FUNCTION_BLOCK FB_Pump_Test EXTENDS FB_TestSuite
VAR_INPUT
END_VAR
VAR_OUTPUT
END_VAR
VAR
END_VAR

Initialize();
EnableTriggersReadyState();
SetFullOutput();
SetZeroOutput();
SetPartialOutput();
DisableOverridesInput();
ClampHighValues();
ClampLowValues();
AutoShutoff();

METHOD AutoShutoff : REFERENCE TO FB_Test
VAR_INPUT
END_VAR
END_METHOD

METHOD ClampHighValues : REFERENCE TO FB_Test
VAR_INPUT
END_VAR
END_METHOD

METHOD ClampLowValues : REFERENCE TO FB_Test
VAR_INPUT
END_VAR
END_METHOD

METHOD DisableOverridesInput : REFERENCE TO FB_Test
VAR_INPUT
END_VAR
END_METHOD

METHOD EnableTriggersReadyState : REFERENCE TO FB_Test
VAR_INPUT
END_VAR
END_METHOD

METHOD Initialize : REFERENCE TO FB_Test
VAR_INPUT
END_VAR
END_METHOD

METHOD SetFullOutput : REFERENCE TO FB_Test
VAR_INPUT
END_VAR
END_METHOD

METHOD SetPartialOutput : REFERENCE TO FB_Test
VAR_INPUT
END_VAR
END_METHOD

METHOD SetZeroOutput : REFERENCE TO FB_Test
VAR_INPUT
END_VAR
END_METHOD

END_FUNCTION_BLOCK

(* stored: Version 1.1.0.1
   POU FB_Pump_Test: Id {cc7fddef-95ee-4c02-b194-8e9ba1f8e8b9}, SpecialFunc None
   Method AutoShutoff: Id {8e297338-e8d4-4626-b306-496e53606749}
   Method ClampHighValues: Id {1e12cea2-fb37-4a81-a7ec-ad5ec57da3d7}
   Method ClampLowValues: Id {40ddc348-1ba2-4960-898f-41f6316e388f}
   Method DisableOverridesInput: Id {5f1db090-b5b7-4034-9130-6e2ef726e213}
   Method EnableTriggersReadyState: Id {659fd9f9-b8b3-497e-93ca-0eafaac5aff0}
   Method Initialize: Id {f37e181c-663a-4cd9-91bb-5da750fbd14e}
   Method SetFullOutput: Id {3f4ac377-9258-4a3e-90d5-f61f7baf06c4}
   Method SetPartialOutput: Id {b3e3f26c-55cd-4ed0-a1a1-cc9a648119ca}
   Method SetZeroOutput: Id {71a8634b-7d56-4624-b60b-e72447314567} *)
